{attribute 'GeneratedUsingTerminal: EK1100-0000-0018'}
{attribute addProperty BoxType "EK1100-0000-0018"}
{attribute addProperty Id "Beckhoff_ELM35xxEK1122Beckhoff_ELM35xxEK1122_0F7152EB2A_0001_ELM3502_0000_0016ELM3502_B416BFEF50A_0002_ELM3502_0000_0017ELM3502_B416BFEF50A_0003_ELM3502_0000_0018ELM3502_B416BFEF50A_0004_ELM3502_0000_0019ELM3502_B416BFEF50A_0005_ELM3504_0000_0016ELM3504_9E251EA472A_0006_ELM3504_0000_0017ELM3504_9E251EA472A_0007_ELM3504_0000_0018ELM3504_9E251EA472A_0008_ELM3504_0000_0019ELM3504_9E251EA472"}
{attribute addProperty CRC "3095678242"}
{attribute addProperty Size "490"}
TYPE Beckhoff_ELM35xx_B8844D22 EXTENDS EK1100_1FC0878B :
STRUCT
	{attribute addProperty Name "Beckhoff_ELM35xxEK1122"}
	Beckhoff_ELM35xxEK1122 : Beckhoff_ELM35xxEK1122_0F7152EB;
	{attribute addProperty Name "A_0001_ELM3502_0000_0016"}
	A_0001_ELM3502_0000_0016 : ELM3502_B416BFEF;
	{attribute addProperty Name "A_0002_ELM3502_0000_0017"}
	A_0002_ELM3502_0000_0017 : ELM3502_B416BFEF;
	{attribute addProperty Name "A_0003_ELM3502_0000_0018"}
	A_0003_ELM3502_0000_0018 : ELM3502_B416BFEF;
	{attribute addProperty Name "A_0004_ELM3502_0000_0019"}
	A_0004_ELM3502_0000_0019 : ELM3502_B416BFEF;
	{attribute addProperty Name "A_0005_ELM3504_0000_0016"}
	A_0005_ELM3504_0000_0016 : ELM3504_9E251EA4;
	{attribute addProperty Name "A_0006_ELM3504_0000_0017"}
	A_0006_ELM3504_0000_0017 : ELM3504_9E251EA4;
	{attribute addProperty Name "A_0007_ELM3504_0000_0018"}
	A_0007_ELM3504_0000_0018 : ELM3504_9E251EA4;
	{attribute addProperty Name "A_0008_ELM3504_0000_0019"}
	A_0008_ELM3504_0000_0019 : ELM3504_9E251EA4;
END_STRUCT
END_TYPE

(* stored: Version 1.2.0.0, ProductVersion 3.1.4024.9
   DUT Beckhoff_ELM35xx_B8844D22: Id {40948b79-0528-4db5-bccb-4abab5bce9ff} *)
